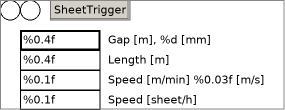
VISUALIZATION _VISU_StartPositionDummy  // 285x110
VAR_IN_OUT
  m_Inst : FB_StartPositionDummy;
END_VAR
    Rectangle (20,30 80x20), "%0.4f", text variable: m_Inst.fSheetGap
        OnMouseClick: write the text variable via Default
    Rectangle (105,70 180x20), "Speed [m/min] %0.03f [m/s]", text variable: m_Inst.fSpeed
    Rectangle (20,70 80x20), "%0.1f", text variable: m_Inst.fSheetSpeed, input disabled if: TRUE
        OnMouseClick: write the text variable via Default
    Rectangle (105,30 180x20), "Gap [m], %d [mm]", text variable: m_Inst.fSheetGap * 1000
    Rectangle (20,50 80x20), "%0.4f", text variable: m_Inst.fSheetLength, input disabled if: TRUE
        OnMouseClick: write the text variable via Default
    Rectangle (105,50 180x20), "Length [m]"
    Ellipse (0,0 20x20), tooltip "Simulation enable"
        toggle m_Inst._bSim
    Button (50,0 80x20), "SheetTrigger", colour toggle: m_Inst.bTrigger
        tap m_Inst.bTrigger
    Rectangle (105,90 180x20), "Speed [sheet/h]"
    Rectangle (20,90 80x20), "%0.1f", text variable: m_Inst.fSheetPerHour, input disabled if: TRUE
        OnMouseClick: write the text variable via Default
    Ellipse (20,0 20x20), tooltip "Simulation auto-trigger"
        toggle m_Inst._bAutoTrigger
END_VISUALIZATION

(* stored: Version 1.1.0.1, ProductVersion 3.1.4024.9
   Visu _VISU_StartPositionDummy: Id {bf231c4c-e11e-4c37-bd97-d2b9e57797fb} *)
